//{attribute 'qualified_only'}
VAR_GLOBAL
	
	//Outputs
	fb_ADS_WATCHDOG_VAC_MRCO_TMO:FB_ADS_WATCHDOG;
	(*ETHERCAT BRIDGE COM STATUS*)
	//0: Other side is in OP state, >0: Error
	{attribute 'TcLinkTo' := 	'TIIB[MRCO_PLC_E04_EL6692]^SYNC Inputs^TxPDO state			 
	'}
	xEcatBridge_TxPDO_state AT %I* : BOOL;
	
	//0: External device connected, 1: External device not connected
	{attribute 'TcLinkTo' := 	'TIIB[MRCO_PLC_E04_EL6692]^SYNC Inputs^External device not connected			 
	'}
	xEcatBridge_External_device_not_connected AT %I* : BOOL;
	
	//0 = Data valid, 1 = Data invalid
	{attribute 'TcLinkTo' := 	'TIIB[MRCO_PLC_E04_EL6692]^WcState^WcState			 
	'}
	xEcatBridge_WcState AT %I* : BOOL;
	
	(*I/O Inputs from TMO Beamline*)
	{attribute 'TcLinkTo' := 	'TIIB[MRCO_PLC_E04_EL6692]^IO Inputs^HUTCH_PLC_NAME			 
	'}
	sHUTCH_PLC_NAME AT %I* : STRING(8);
	
	{attribute 'TcLinkTo' := 	'TIIB[MRCO_PLC_E04_EL6692]^IO Inputs^TMO_ROUGH1_VRC_01_OPEN_LS			 
	'}
	xTMO_ROUGH1_VRC_01_OPEN_LS AT %I* : BOOL;
	
	{attribute 'TcLinkTo' := 	'TIIB[MRCO_PLC_E04_EL6692]^IO Inputs^TMO_ROUGH2_VRC_01_OPEN_LS			 
	'}
	xTMO_ROUGH2_VRC_01_OPEN_LS AT %I* : BOOL;
	
	
	(*I/O Outputs to TMO Beamline*)
	{attribute 'TcLinkTo' := 	'TIIB[MRCO_PLC_E04_EL6692]^IO Outputs^ENDSTATION_PLC_NAME			 
	'}
	sENDSTATION_PLC_NAME AT %Q* : STRING(8):= 'MRCO';
	
	{attribute 'TcLinkTo' := 	'TIIB[MRCO_PLC_E04_EL6692]^IO Outputs^IP1_ROUGH_VRC_01_OPEN_LS			 
	'}
	xIP1_ROUGH_VRC_01_OPEN_LS AT %Q* : BOOL;
	
	{attribute 'TcLinkTo' := 	'TIIB[MRCO_PLC_E04_EL6692]^IO Outputs^IP1_ROUGH_VRC_02_OPEN_LS			 
	'}
	xIP1_ROUGH_VRC_02_OPEN_LS AT %Q* : BOOL;
	
	{attribute 'TcLinkTo' := 	'TIIB[MRCO_PLC_E04_EL6692]^IO Outputs^IP1_ROUGH_VRC_03_OPEN_LS			 
	'}
	xIP1_ROUGH_VRC_03_OPEN_LS AT %Q* : BOOL;
	
	{attribute 'TcLinkTo' := 	'TIIB[MRCO_PLC_E04_EL6692]^IO Outputs^IP1_TURBOS_ALL_AtSpd			 
	'}
	{attribute 'pytmc' := '
		pv: PLC:MRCO:VAC:IP1_TURBOS_ALL_ATSPD
		io:i
	'}
	xIP1_TURBOS_ALL_AtSpd AT %Q* : BOOL;
	
	{attribute 'TcLinkTo' := 	'TIIB[MRCO_PLC_E04_EL6692]^IO Outputs^IP1_MAIN_xAT_VAC			 
	'}
	xIP1_MAIN_xAT_VAC AT %Q* : BOOL;
	
	{attribute 'TcLinkTo' := 	'TIIB[MRCO_PLC_E04_EL6692]^IO Outputs^IP1_MAIN_xPRESS_OK			 
	'}
	xIP1_MAIN_xPRESS_OK AT %Q* : BOOL;
	
	{attribute 'TcLinkTo' := 	'TIIB[MRCO_PLC_E04_EL6692]^IO Outputs^IP1_MAIN_rPRESS			 
	'}
	rIP1_MAIN_rPRESS AT %Q* : REAL;
	
	{attribute 'TcLinkTo' := 	'TIIB[MRCO_PLC_E04_EL6692]^IO Outputs^IP1_HV_SAFETY_ENABLE			 
	'}
	xIP1_HV_SAFETY_ENABLE AT %Q* : BOOL;
	
	
	(*ISEG HV Crate Safety Loop*)
	{attribute 'TcLinkTo' := 	'TIIB[MRCO_PLC_E09_EL2794]^Channel 1^Output			 
	'}
	{attribute 'pytmc' := '
		pv: PLC:MRCO:VAC:HV_SAFETY_ENABLE
		io:i
	'}
	xHighVoltageSafteyLoopEnable AT %Q* : BOOL := FALSE; (*When Enables the High voltage Saftey loop is closed and HV can start.*)
END_VAR

(* stored: Version 1.1.0.1, ProductVersion 3.1.4024.2
   GVL GVL_PLC_Interfaces: Id {2bd01e0b-5a43-46af-b534-be253d3d7c4a} *)
